FUNCTION_BLOCK PUBLIC FB_DecoratorCheese EXTENDS FB_Decorator
VAR_INPUT
END_VAR
VAR_OUTPUT
END_VAR
VAR
END_VAR

METHOD GetDescription : STRING
IF (SUPER^.ipSideOrder <> 0) THEN
	GetDescription := CONCAT (SUPER^.ipSideOrder.GetDescription(), ' - Cheese');
END_IF
END_METHOD

METHOD GetPrice : LREAL
IF (SUPER^.ipSideOrder <> 0) THEN
	GetPrice := SUPER^.ipSideOrder.GetPrice() + 1.1;
END_IF
END_METHOD

END_FUNCTION_BLOCK

(* stored: Version 1.1.0.1, ProductVersion 3.1.4022.16
   POU FB_DecoratorCheese: Id {9ad8c55b-8edd-47dc-b2f2-450a6798519a}, SpecialFunc None
   Method GetDescription: Id {982907fa-22f1-4520-92dd-1be191c4fdf4}
   Method GetPrice: Id {bf93a2ab-e89a-430c-9a8f-8bbb7796ec9a} *)
